TYPE ST_INSTANCE_CTRL :
STRUCT
  Cmd     : E_INSTANCE_CMD;
END_STRUCT
END_TYPE

(* stored: Version 1.1.0.1, ProductVersion 3.1.4026.13
   DUT ST_INSTANCE_CTRL: Id {bc5c1f71-6eb7-44f0-9eb2-ac0cd0afc11c} *)
